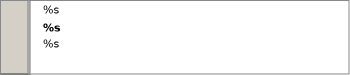
VISUALIZATION Uc_EventLogEntry  // 350x75
    Group (0,0 350x75), invisible if: stVisu.nIdx < 0
        Rectangle (0,0 350x75), colour toggle: stVisu.nIdx = nSelectId
            p2167032090: stVisu.nPriorityColor-16#C8000000
            OnMouseClick: execute { nSelectId := stVisu.nIdx; }
        Rectangle (40,2 300x15), "%s", text variable: stVisu.sRaiseInfo
        Rectangle (40,20 300x16), "%s", text variable: stVisu.sPosition
        Rectangle (40,36 300x32), "%s", text variable: stVisu.sDescription
        Rectangle (0,0 350x75)
            OnMouseClick: execute { nSelectId := stVisu.nIdx; }
        Rectangle (0,0 10x75), colour variable: stVisu.nPriorityColor
            p3450524324: stVisu.nPriorityColor
        Button (0,0 30x75), invisible if: NOT (stVisu.nIdx = nSelectId)
            p2175578022: stVisu.nPriorityColor
            tap bQuit
END_VISUALIZATION

(* stored: Version 1.1.0.1
   Visu Uc_EventLogEntry: Id {efb8db71-d947-43bd-8f1f-67019412fbb9} *)
